// Writes a uint64 field value, without a tag, to the stream.
FUNCTION F_WriteUInt64 : HRESULT
VAR_IN_OUT
    aBuffer : ARRAY [*] OF BYTE;
    stState : ST_WriterInternalState;
END_VAR
VAR_INPUT
    nValue : ULINT;
END_VAR
VAR
END_VAR

F_WriteUInt64 := F_WriteRawVarint64(aBuffer, stState, nValue);

END_FUNCTION

(* stored: Version 1.1.0.1
   POU F_WriteUInt64: Id {1c0ef302-717f-4938-884e-42b4d492e8ae}, SpecialFunc None *)
